//     Term 9 (APS4322-7000)/APS Outputs/Current Q 1X0 <-> Data Pointer/QCurrentSetPoints[6]
//     Term 9 (APS4322-7000)/APS Outputs/Current Q 1X1 <-> Data Pointer/QCurrentSetPoints[7]
//     Term 9 (APS4322-7000)/APS Outputs/Current Q 1X2 <-> Data Pointer/QCurrentSetPoints[8]
//     Term 9 (APS4322-7000)/APS Outputs/Current Q 2X0 <-> Data Pointer/QCurrentSetPoints[12]
//     Term 9 (APS4322-7000)/APS Outputs/Current Q 2X1 <-> Data Pointer/QCurrentSetPoints[13]
//     Term 9 (APS4322-7000)/APS Outputs/Current Q 2X2 <-> Data Pointer/QCurrentSetPoints[14]
//     Term 9 (APS4322-7000)/APS Outputs/Current Q 3X0 <-> Data Pointer/QCurrentSetPoints[18]
//     Term 9 (APS4322-7000)/APS Outputs/Current Q 3X1 <-> Data Pointer/QCurrentSetPoints[19]
//     Term 9 (APS4322-7000)/APS Outputs/Current Q 3X2 <-> Data Pointer/QCurrentSetPoints[20]
//     Term 9 (APS4322-7000)/APS Outputs/Current Q 0Y0 <-> Data Pointer/QCurrentSetPoints[3]
//     Term 9 (APS4322-7000)/APS Outputs/Current Q 0Y1 <-> Data Pointer/QCurrentSetPoints[4]
//     Term 9 (APS4322-7000)/APS Outputs/Current Q 0Y2 <-> Data Pointer/QCurrentSetPoints[5]
//     Term 9 (APS4322-7000)/APS Outputs/Current Q 1Y0 <-> Data Pointer/QCurrentSetPoints[9]
//     Term 9 (APS4322-7000)/APS Outputs/Current Q 1Y1 <-> Data Pointer/QCurrentSetPoints[10]
//     Term 9 (APS4322-7000)/APS Outputs/Current Q 1Y2 <-> Data Pointer/QCurrentSetPoints[11]
//     Term 9 (APS4322-7000)/APS Outputs/Current Q 2Y0 <-> Data Pointer/QCurrentSetPoints[15]
//     Term 9 (APS4322-7000)/APS Outputs/Current Q 2Y1 <-> Data Pointer/QCurrentSetPoints[16]
//     Term 9 (APS4322-7000)/APS Outputs/Current Q 2Y2 <-> Data Pointer/QCurrentSetPoints[17]
//     Term 9 (APS4322-7000)/APS Outputs/Current Q 3Y0 <-> Data Pointer/QCurrentSetPoints[21]
//     Term 9 (APS4322-7000)/APS Outputs/Current Q 3Y1 <-> Data Pointer/QCurrentSetPoints[22]
//     Term 9 (APS4322-7000)/APS Outputs/Current Q 3Y2 <-> Data Pointer/QCurrentSetPoints[23]
//     Term 9 (APS4322-7000)/APS Outputs/PhiE 0X0 <-> Data Pointer/PhiSetPoints[0]
//     Term 9 (APS4322-7000)/APS Outputs/PhiE 0X1 <-> Data Pointer/PhiSetPoints[1]
//     Term 9 (APS4322-7000)/APS Outputs/PhiE 0X2 <-> Data Pointer/PhiSetPoints[2]
//     Term 9 (APS4322-7000)/APS Outputs/PhiE 1X0 <-> Data Pointer/PhiSetPoints[6]
//     Term 9 (APS4322-7000)/APS Outputs/PhiE 1X1 <-> Data Pointer/PhiSetPoints[7]
//     Term 9 (APS4322-7000)/APS Outputs/PhiE 1X2 <-> Data Pointer/PhiSetPoints[8]
//     Term 9 (APS4322-7000)/APS Outputs/PhiE 2X0 <-> Data Pointer/PhiSetPoints[12]
//     Term 9 (APS4322-7000)/APS Outputs/PhiE 2X1 <-> Data Pointer/PhiSetPoints[13]
//     Term 9 (APS4322-7000)/APS Outputs/PhiE 2X2 <-> Data Pointer/PhiSetPoints[14]
//     Term 9 (APS4322-7000)/APS Outputs/PhiE 3X0 <-> Data Pointer/PhiSetPoints[18]
//     Term 9 (APS4322-7000)/APS Outputs/PhiE 3X1 <-> Data Pointer/PhiSetPoints[19]
//     Term 9 (APS4322-7000)/APS Outputs/PhiE 3X2 <-> Data Pointer/PhiSetPoints[20]
//     Term 9 (APS4322-7000)/APS Outputs/PhiE 0Y0 <-> Data Pointer/PhiSetPoints[3]
//     Term 9 (APS4322-7000)/APS Outputs/PhiE 0Y1 <-> Data Pointer/PhiSetPoints[4]
//     Term 9 (APS4322-7000)/APS Outputs/PhiE 0Y2 <-> Data Pointer/PhiSetPoints[5]
//     Term 9 (APS4322-7000)/APS Outputs/PhiE 1Y0 <-> Data Pointer/PhiSetPoints[9]
//     Term 9 (APS4322-7000)/APS Outputs/PhiE 1Y1 <-> Data Pointer/PhiSetPoints[10]
//     Term 9 (APS4322-7000)/APS Outputs/PhiE 1Y2 <-> Data Pointer/PhiSetPoints[11]
//     Term 9 (APS4322-7000)/APS Outputs/PhiE 2Y0 <-> Data Pointer/PhiSetPoints[15]
//     Term 9 (APS4322-7000)/APS Outputs/PhiE 2Y1 <-> Data Pointer/PhiSetPoints[16]
//     Term 9 (APS4322-7000)/APS Outputs/PhiE 2Y2 <-> Data Pointer/PhiSetPoints[17]
//     Term 9 (APS4322-7000)/APS Outputs/PhiE 3Y0 <-> Data Pointer/PhiSetPoints[21]
//     Term 9 (APS4322-7000)/APS Outputs/PhiE 3Y1 <-> Data Pointer/PhiSetPoints[22]
//     Term 9 (APS4322-7000)/APS Outputs/PhiE 3Y2 <-> Data Pointer/PhiSetPoints[23]
//     Term 9 (APS4322-7000)/Term 10 (APS4322-5000)/FB Inputs/A{0..8 step 2} X-Field <-> Data Pointer/HallSensorFieldsXYZ[{0..12 step 3}]  (5 links)
//     Term 9 (APS4322-7000)/Term 10 (APS4322-5000)/FB Inputs/A{0..8 step 2} Y-Field <-> Data Pointer/HallSensorFieldsXYZ[{1..13 step 3}]  (5 links)
//     Term 9 (APS4322-7000)/Term 10 (APS4322-5000)/FB Inputs/A{0..8 step 2} Z-Field <-> Data Pointer/HallSensorFieldsXYZ[{2..14 step 3}]  (5 links)
//     Term 9 (APS4322-7000)/Term 10 (APS4322-5000)/FB Inputs/B{1..9 step 2} X-Field <-> Data Pointer/HallSensorFieldsXYZ[{15..27 step 3}]  (5 links)
//     Term 9 (APS4322-7000)/Term 10 (APS4322-5000)/FB Inputs/B{1..9 step 2} Y-Field <-> Data Pointer/HallSensorFieldsXYZ[{16..28 step 3}]  (5 links)
//     Term 9 (APS4322-7000)/Term 10 (APS4322-5000)/FB Inputs/B{1..9 step 2} Z-Field <-> Data Pointer/HallSensorFieldsXYZ[{17..29 step 3}]  (5 links)
//     Term 9 (APS4322-7000)/Term 10 (APS4322-5000)/FB Inputs/C{0..8 step 2} X-Field <-> Data Pointer/HallSensorFieldsXYZ[{30..42 step 3}]  (5 links)
//     Term 9 (APS4322-7000)/Term 10 (APS4322-5000)/FB Inputs/C{0..8 step 2} Y-Field <-> Data Pointer/HallSensorFieldsXYZ[{31..43 step 3}]  (5 links)
//     Term 9 (APS4322-7000)/Term 10 (APS4322-5000)/FB Inputs/C{0..8 step 2} Z-Field <-> Data Pointer/HallSensorFieldsXYZ[{32..44 step 3}]  (5 links)
//     Term 9 (APS4322-7000)/Term 10 (APS4322-5000)/FB Inputs/D{1..9 step 2} X-Field <-> Data Pointer/HallSensorFieldsXYZ[{45..57 step 3}]  (5 links)
//     Term 9 (APS4322-7000)/Term 10 (APS4322-5000)/FB Inputs/D{1..9 step 2} Y-Field <-> Data Pointer/HallSensorFieldsXYZ[{46..58 step 3}]  (5 links)
//     Term 9 (APS4322-7000)/Term 10 (APS4322-5000)/FB Inputs/D{1..9 step 2} Z-Field <-> Data Pointer/HallSensorFieldsXYZ[{47..59 step 3}]  (5 links)
//     Term 9 (APS4322-7000)/Term 10 (APS4322-5000)/FB Inputs/E{0..8 step 2} X-Field <-> Data Pointer/HallSensorFieldsXYZ[{60..72 step 3}]  (5 links)
//     Term 9 (APS4322-7000)/Term 10 (APS4322-5000)/FB Inputs/E{0..8 step 2} Y-Field <-> Data Pointer/HallSensorFieldsXYZ[{61..73 step 3}]  (5 links)
//     Term 9 (APS4322-7000)/Term 10 (APS4322-5000)/FB Inputs/E{0..8 step 2} Z-Field <-> Data Pointer/HallSensorFieldsXYZ[{62..74 step 3}]  (5 links)
//     Term 9 (APS4322-7000)/Term 10 (APS4322-5000)/FB Inputs/F{1..9 step 2} X-Field <-> Data Pointer/HallSensorFieldsXYZ[{75..87 step 3}]  (5 links)
//     Term 9 (APS4322-7000)/Term 10 (APS4322-5000)/FB Inputs/F{1..9 step 2} Y-Field <-> Data Pointer/HallSensorFieldsXYZ[{76..88 step 3}]  (5 links)
//     Term 9 (APS4322-7000)/Term 10 (APS4322-5000)/FB Inputs/F{1..9 step 2} Z-Field <-> Data Pointer/HallSensorFieldsXYZ[{77..89 step 3}]  (5 links)
//     Term 9 (APS4322-7000)/Term 10 (APS4322-5000)/FB Inputs/G{0..8 step 2} X-Field <-> Data Pointer/HallSensorFieldsXYZ[{90..102 step 3}]  (5 links)
//     Term 9 (APS4322-7000)/Term 10 (APS4322-5000)/FB Inputs/G{0..8 step 2} Y-Field <-> Data Pointer/HallSensorFieldsXYZ[{91..103 step 3}]  (5 links)
//     Term 9 (APS4322-7000)/Term 10 (APS4322-5000)/FB Inputs/G{0..8 step 2} Z-Field <-> Data Pointer/HallSensorFieldsXYZ[{92..104 step 3}]  (5 links)
//     Term 9 (APS4322-7000)/Term 10 (APS4322-5000)/FB Inputs/H{1..9 step 2} X-Field <-> Data Pointer/HallSensorFieldsXYZ[{105..117 step 3}]  (5 links)
//     Term 9 (APS4322-7000)/Term 10 (APS4322-5000)/FB Inputs/H{1..9 step 2} Y-Field <-> Data Pointer/HallSensorFieldsXYZ[{106..118 step 3}]  (5 links)
//     Term 9 (APS4322-7000)/Term 10 (APS4322-5000)/FB Inputs/H{1..9 step 2} Z-Field <-> Data Pointer/HallSensorFieldsXYZ[{107..119 step 3}]  (5 links)
//     Term 9 (APS4322-7000)/Term 10 (APS4322-5000)/FB Inputs/I{0..8 step 2} X-Field <-> Data Pointer/HallSensorFieldsXYZ[{120..132 step 3}]  (5 links)
//     Term 9 (APS4322-7000)/Term 10 (APS4322-5000)/FB Inputs/I{0..8 step 2} Y-Field <-> Data Pointer/HallSensorFieldsXYZ[{121..133 step 3}]  (5 links)
//     Term 9 (APS4322-7000)/Term 10 (APS4322-5000)/FB Inputs/I{0..8 step 2} Z-Field <-> Data Pointer/HallSensorFieldsXYZ[{122..134 step 3}]  (5 links)
//     Term 9 (APS4322-7000)/Term 10 (APS4322-5000)/FB Inputs/J{1..9 step 2} X-Field <-> Data Pointer/HallSensorFieldsXYZ[{135..147 step 3}]  (5 links)
//     Term 9 (APS4322-7000)/Term 10 (APS4322-5000)/FB Inputs/J{1..9 step 2} Y-Field <-> Data Pointer/HallSensorFieldsXYZ[{136..148 step 3}]  (5 links)
//     Term 9 (APS4322-7000)/Term 10 (APS4322-5000)/FB Inputs/J{1..9 step 2} Z-Field <-> Data Pointer/HallSensorFieldsXYZ[{137..149 step 3}]  (5 links)
//     Term 9 (APS4322-7000)/Term 10 (APS4322-5000)/FB Inputs/Status <-> Data Pointer/FeedbackStatus

CONFIGURATION Plc
    RESOURCE PLC ON TwinCAT3
        TASK PlcTask(INTERVAL := T#10ms, PRIORITY := 6);
        PROGRAM MAIN WITH PlcTask : MAIN;
    END_RESOURCE
END_CONFIGURATION

// ---- THREADs/Example Product Data/ST_ProductDataA.TcDUT
TYPE ST_ProductDataA :
STRUCT
	nQuality : UINT;
	bGoodProduct : BOOL;
END_STRUCT
END_TYPE

// ---- THREADs/Example Product Data/I_ProductDataA.TcIO
INTERFACE I_ProductDataA EXTENDS I_XP_ProductData

{attribute 'monitoring':='call'}
PROPERTY Data : REFERENCE TO ST_ProductDataA
GET
END_GET
END_PROPERTY

END_INTERFACE

// ---- THREADs/MAIN.TcPOU
PROGRAM MAIN
VAR CONSTANT
	cCtsXpMovers : UINT := 3;	
	cCtsXpTracks : UINT := 6;	
	//Unique station identification 
	S_INFEED1 	: STRING := 'Station A';
	S_OUTFEED1 	: STRING := 'Station D';
	//Groupe station identification 
	G_PROCESS	: STRING := 'Groupe Process';
END_VAR
VAR
	bInitDone 			: BOOL;
	bEnable				: BOOL;
	bDisable, bReset	: BOOL;
	bSetSettings 		: BOOL := TRUE;
	
	(* XPlanar System - 1 per associated XPlanar 
		The system is the container and organizer for all subsequent XPlanar objects. All objects are registered with this system*)
	fbXpSystem : FB_XP_System;
	ipXPlanarPLC : I_XP_System_PLC := fbXpSystem; 
	
	(* XPlanar Collision Avoidance Groupe - 1 per associated XPlanar 
		The Planar group is a software object that prevents collisions between Planar movers as well as collisions of Planar movers with the boundary of 
		the stator area on the two-dimensional XPlanar stator area. To do this, the 2D areas of all objects in the group are blocked. When a motion command 
		is transferred to a mover, the required area is requested from the Planar group and the motion command is rejected if this area would collide 
		with already reserved areas. If the motion command can be executed, the area is added to the set of reserved area and blocked accordingly. *)
	fbXpGroup : FB_XP_Group
									(ipSystem			:= fbXpSystem);
	(* XPlanar Environment - 1 per associated XPlanar 
		The Planar environment is a software object that represents the two-dimensional XPlanar stator surface. Together with Planar movers in a group, 
		it prevents collisions of the movers with the edge of the surface. *)
	fbXpEnvironment : FB_XP_Environment
									(ipSystem			:= fbXpSystem);	
	
	(* XPlanar mover - n per associated XPlanar. Can be instantiated as an array and/or individually
		The Planar mover is a software object that represents an XPlanar mover. It summarizes the state of the real mover (position, velocity, etc.) 
		for the user. In addition, the user has the possibility to influence or control the state of the real mover via the Planar mover. *)								
	aMovers : ARRAY[1..cCtsXpMovers] OF FB_XP_Mover[
								 	(ipSystem			:= fbXpSystem),
								 	(ipSystem			:= fbXpSystem),
								 	(ipSystem			:= fbXpSystem)];

	(* XPlanar track - n per associated XPlanar. Can be instantiated as an array and/or individually
		The Planar track is a software object that represents a (virtual) one-dimensional path on the two-dimensional XPlanar stator surface. 
		Several Planar movers can be lined up and moved on this path. Collisions are prevented by keeping a preset distance between the movers. *)		
	aTracks : ARRAY[1..cCtsXpTracks] OF FB_XP_Track[
								 	(ipSystem			:= fbXpSystem),
								 	(ipSystem			:= fbXpSystem),
								 	(ipSystem			:= fbXpSystem),
								 	(ipSystem			:= fbXpSystem),
								 	(ipSystem			:= fbXpSystem),
								 	(ipSystem			:= fbXpSystem)];

	(* XPlanar station - n per associated XPlanar. Can be instantiated as an array and/or individually
		The stations are the main component of the application. As soon as the system has been started up and all movers are on the track, the movers are only sent from one station to the next.
		Parameters:
			xPos, yPos 			= Absolute position of the station on the xPlanar.
			ipAccocietedTrack 	= The track on which the station is located. If the XY position is not on this track, the next possible track position is assumed on this track.
								  Can be set to 0. In this case, the closest track to the coordinates is automatically used. 
								  If the station is very close to a transition, it may still be interesting to enter the exact track here.		
			sUniqueName 		= Unique name that may only exist once.
			sTargetGroup 		= A name for a group to which this station belongs. Important for redundant stations	*)	
	fbStationA : FB_XP_Station(ipSystem 			:= fbXpSystem,
									ipAccocietedTrack 	:= 0,// =closest track
									sUniqueName			:= S_INFEED1,
									sTargetGroup		:= '',
									nMoverQueueSize		:= 1,
									xPos				:= 100,
									yPos				:= 540);
									
	fbStationB 		: FB_XP_Station(ipSystem 			:= fbXpSystem,
									ipAccocietedTrack 	:= 0, // =closest track
									sUniqueName 		:= '',
									sTargetGroup		:= G_PROCESS,
									nMoverQueueSize		:= 1,
									xPos				:= 600,
									yPos				:= 600);	
		
	fbStationC 		: FB_XP_Station(ipSystem 			:= fbXpSystem,
									ipAccocietedTrack 	:= 0, // =closest track
									sUniqueName 		:= '',
									sTargetGroup		:= G_PROCESS,
									nMoverQueueSize		:= 1,
									xPos				:= 600,
									yPos				:= 120);						
										
	fbStationD 		: FB_XP_Station(ipSystem 			:= fbXpSystem,
									ipAccocietedTrack 	:= 0, // =closest track
									sUniqueName 		:= S_OUTFEED1,
									sTargetGroup		:= '',
									nMoverQueueSize		:= 2,
									xPos				:= 120,
									yPos				:= 400);	
											
	fbStationD_ChangeGap 		: FB_XP_Station(ipSystem := fbXpSystem,
									ipAccocietedTrack 	:= 0, // =closest track
									sUniqueName 		:= '',
									sTargetGroup		:= '',
									nMoverQueueSize		:= 1,
									xPos				:= 188,//120,125
									yPos				:= 90);						
													
	(*Processing station*)								
	fbStationCLowerZ : FB_Station_LowerZForce(ipStation := fbStationC);	
	fbStationBExternalSetpoint : FB_Station_ExternalSetpoint(ipStation := fbStationB);							
									
	(* EtherCAt diagnostics - TC3_Eventlogger
	This function block instance scans the entire EtherCat master. 
	Each EtherCat slave device is recognized and a message is written to the TC3_Eventlogger as soon as an unwanted state occurs.*)
	//	fbEtherCatDiagLAN3 : FB_EtherCatMasterDiag;
	//	fbEtherCatDiagLAN4 : FB_EtherCatMasterDiag;
END_VAR

//Example ConfigTrack
VAR
	bDoConfigTrackC 		: BOOL := TRUE;
	nSeqConfigTrack 		: UINT;
	fbTrackFeedback 		: MC_PlanarFeedback;	
	posStart, posEnd 		: PositionXYC; 
END_VAR

//Example SimulationMode
VAR
	bStartSimulation,bStopSimulation : BOOL;
END_VAR

//Example Manual Interaction with process outside XPlanar
VAR
	bToUpstreamProcessCanStart 		: BOOL; //Requestet cts of mover are in station. Example: rototer can start to place prodcts
	bFromUpsreamProcessIsFinish 	: BOOL; //The upstream process can set this bool if the process is finish and the mover can leave the station
	sFromUpstreamTagedStation		: STRING; //The Upstream can chose where the movers should go next
END_VAR

IF NOT bInitDone THEN
 	ipXPlanarPLC.Initialize();
	bInitDone := ipXPlanarPLC.Initialized;
	RETURN;
END_IF

IF bEnable AND ipXPlanarPLC.Disabled THEN
	bEnable := FALSE;
	ipXPlanarPLC.Enable();
	bSetSettings := TRUE; // Write Settings once
END_IF

IF bDisable OR bReset THEN
	bDisable := FALSE; bReset := FALSE;
	ipXPlanarPLC.Disable();
END_IF

IF bStartSimulation AND ipXPlanarPLC.Enabled THEN
	bStartSimulation := FALSE;
	fbStationA.SimulationStart(fProcessDuration := 0.1, sTargetStation := G_PROCESS); //Groupe
	fbStationD.SimulationStart(fProcessDuration := 0.5, sTargetStation := S_INFEED1); //Exact Station
	
	//fbStationB.SimulationStart(fProcessDuration := 1.0, sTargetStation := S_OUTFEED1); 
	fbStationBExternalSetpoint.TargetStation := S_OUTFEED1;	
	
	//fbStationC.SimulationStart(fProcessDuration := 1.0, sTargetStation := S_OUTFEED1);
	fbStationCLowerZ.TargetStation := S_OUTFEED1;
END_IF

IF bStopSimulation THEN
	bStopSimulation := FALSE;
	fbStationA.SimulationStop();
	fbStationB.SimulationStop();
	fbStationC.SimulationStop();
	fbStationD.SimulationStop();
END_IF


//Calculate setting each cycle
IF ipXPlanarPLC.Enabled THEN
	//Movement to the station is only permitted if the track is free. 
	//This serves to prevent collisions as only the gap is not sufficient here
	fbStationB.ReadyToRecvMovers := fbStationB.AccocietedTrack.CtsMoversOnTrack = 0;
	fbStationC.ReadyToRecvMovers := fbStationC.AccocietedTrack.CtsMoversOnTrack = 0;
ELSE
	fbStationB.ReadyToRecvMovers := FALSE;
	fbStationC.ReadyToRecvMovers := FALSE;
END_IF


//Do settings once at eanbling
IF bSetSettings THEN
	bSetSettings := FALSE;
	
	//TODO: The very first time the system is started up, the mover does not yet have a target. 
	//The default target defined in the CHALET_Xplanar/parameter list is entered. You should adjust the defaulttrged 

	//Set Mover Velocity, Acc, Dec, Jerk once. The station will override this settings
	aMovers[1].SetDynConstraint_Path(200,1900,1900,20000);
	aMovers[2].SetDynConstraint_Path(200,1900,1900,20000);
	aMovers[3].SetDynConstraint_Path(200,1900,1900,20000);
	
	//"In Position" is set 5mm earlier
	fbStationA.TargetPosWindow := 5.0;
	
	//The mover gets this targed gap asson he leves the station
	fbStationA.MoverGapAtExit := 300.0;
	fbStationD_ChangeGap.MoverGapAtExit := 190.0;
	
	fbStationB.MoverVelocityAtExit := 2000;	
	fbStationB.MoverAccAtExit := MC_MAXIMUM;
	fbStationB.MoverDecAtExit := MC_MAXIMUM;
	
	fbStationC.MoverVelocityAtExit := 2000;	
	fbStationC.MoverAccAtExit := MC_DEFAULT;
END_IF


PRG_Example_ProductData_Simple();


(* Update is called at the end of the program *)
ipXPlanarPLC.Update();
fbStationCLowerZ.Update();
fbStationBExternalSetpoint.Update();
//fbEtherCatDiagLAN3.Update();
//fbEtherCatDiagLAN4.Update();

METHOD Example_ManualConfigTrack : BOOL
(* Instead of the track being initialized in the track object, 
   the track progression can also be set here in the PLC. 
   To change values in the PLC, the track must be disabled (system is disabled) and the value to be changed must not be described in the object. 
*)
IF bDoConfigTrackC AND xPlanarPLC.Disabled THEN
	CASE nSeqConfigTrack OF
		0: //Clears the geometric information of the Planar Track.
			fbTrackC.PlanarTrack.Clear(fbTrackFeedback);
			nSeqConfigTrack := nSeqConfigTrack + 1;
		
		1: //Wait for command finished successfully
			IF fbTrackFeedback.Done THEN
				nSeqConfigTrack := nSeqConfigTrack + 1;
			END_IF
			
		2: //Sets the other Planar Tracks endpoint as start point of this Planar Track, transition is smooth. The other Planar Track is blocked for further changes (until it is cleared).
			fbTrackC.PlanarTrack.StartFromTrack(track := fbTrackA.PlanarTrack, commandFeedback := fbTrackFeedback);
			nSeqConfigTrack := nSeqConfigTrack + 1;
		
		3: //Wait for command finished successfully
			IF fbTrackFeedback.Done THEN
				nSeqConfigTrack := nSeqConfigTrack + 1;
			END_IF
			
		4: //Appends a line to the Planar Track.
			posStart.SetValuesXYC(840,480,0);
			posEnd.SetValuesXYC(840,240,0);
			fbTrackC.PlanarTrack.AppendLine(start := posStart, end := posEnd, commandFeedback := fbTrackFeedback);
			nSeqConfigTrack := nSeqConfigTrack + 1;					

		5: //Wait for command finished successfully
			IF fbTrackFeedback.Done THEN
				nSeqConfigTrack := nSeqConfigTrack + 1;
			END_IF
			
		6: //Appends a smooth transition from the end of this Planar Track to the other Planar Tracks start point. The Planar Track is blocked for further changes (until it is cleared).
			fbTrackC.PlanarTrack.EndAtTrack(track := fbTrackA.PlanarTrack, commandFeedback := fbTrackFeedback);
			nSeqConfigTrack := nSeqConfigTrack + 1;
		
		7: //Wait for command finished successfully
			IF fbTrackFeedback.Done THEN
				nSeqConfigTrack := nSeqConfigTrack + 1;
			END_IF		
		
		8: //Done
			bDoConfigTrackC := FALSE;
			nSeqConfigTrack := 0;
	END_CASE
	fbTrackFeedback.Update(); 
END_IF
END_METHOD

METHOD Example_ManualInteractionWithProcess : BOOL
(* Example: Interaction with process outside XPlanar 
   only works when the simulation is switched off
*)

//Requestet cts of mover are in station. Example: rototer can start to place prodcts
bToUpstreamProcessCanStart := xPlanarPLC.Station(S_INFEED1).MoversInPlace;

//The upstream process can set this bool if the process is finish and the mover can leave the station
bFromUpsreamProcessIsFinish := bFromUpsreamProcessIsFinish;

//The Upstream can chose where the movers should go next
//A group is specified here that contains several different. equivalent stations
sFromUpstreamTagedStation := G_OUTFEED;

IF bFromUpsreamProcessIsFinish AND bToUpstreamProcessCanStart AND xPlanarPLC.Enabled THEN
	bFromUpsreamProcessIsFinish := FALSE;
	xPlanarPLC.Station(S_INFEED1).SendMoversToStation(sFromUpstreamTagedStation);
END_IF
END_METHOD

END_PROGRAM

// ---- THREADs/FB_Station_LowerZForce.TcPOU
FUNCTION_BLOCK FB_Station_LowerZForce EXTENDS FB_CH_Object
VAR
	ipStation : I_XP_Station_PLC;
	nSeq : UINT;
	fbTon : TON;
	ipMoverInStation : I_XP_Mover_PLC;
	bFromUpstreamProcessIsFinish: BOOL := TRUE;
	sTargetStation : STRING; //the mover gets this as next target
END_VAR

METHOD FB_init : BOOL
VAR_INPUT
	bInitRetains : BOOL; // if TRUE, the retain variables are initialized (warm start / cold start)
	bInCopyCode : BOOL;  // if TRUE, the instance afterwards gets moved into the copy code (online change)
	
	ipStation : I_XP_Station_PLC;
	
END_VAR
VAR
	fbGetCurTaskIdx  : GETCURTASKINDEX;
END_VAR
THIS^.ipStation := ipStation;
END_METHOD

{attribute 'monitoring':='call'}
 //the mover gets this as next target
PROPERTY TargetStation : STRING
GET
TargetStation := sTargetStation;
END_GET
SET
sTargetStation := TargetStation;
END_SET
END_PROPERTY

METHOD Update : HRESULT
VAR
	refPlanarTrack : REFERENCE TO MC_PlanarTrack;
END_VAR
IF ipStation = 0 THEN
	RETURN; // ERROR
END_IF

IF ipStation.System.Disabled THEN
	nSeq := 0;
END_IF

//The simulation (automatic retransmission of a mover after a fixed time) is stopped for this station
ipStation.SimulationStop();

CASE nSeq OF 

	0: //wait for mover
		IF ipStation.MoversInPlace THEN
			//receive the foremost mover in the station (if there is more than one mover in the station)
			ipMoverInStation := ipStation.MoversInQueue[0];
			nSeq := 1;
		END_IF
		
	1: //Z = 0
		ipMoverInStation.LowerToUnknownLevel();
		nSeq := 2;				

	2: // wait until lowering is finish
		IF ipMoverInStation.Feedback.Done THEN
			fbTon.IN := FALSE;
			nSeq := 3;	
		END_IF
		
	3: //Delay 5s
		fbTon.IN := TRUE;
		IF fbTon.q THEN
			nSeq := 4;	
		END_IF			

	4: //Lift
		ipMoverInStation.LiftFromUnknownLevel();
		nSeq := 5;				

	5: // wait until lifting is finish
		//The upstream process can set this bool if the process is finish and the mover can leave the station
		bFromUpstreamProcessIsFinish := bFromUpstreamProcessIsFinish;

		fbTon.IN := TRUE;
		IF fbTon.q AND bFromUpstreamProcessIsFinish THEN
			nSeq := 100;	
		END_IF

		
	100: // send movers away to next target station or groupe. If no target exist, wait in this step
		IF sTargetStation <> '' THEN
			ipStation.SendMoversToStation(THIS^.sTargetStation);
			nSeq := 0;	
		END_IF

	
END_CASE
fbTon(PT:= T#5S);
END_METHOD

END_FUNCTION_BLOCK

// ---- THREADs/FB_Station_ExternalSetpoint.TcPOU
FUNCTION_BLOCK FB_Station_ExternalSetpoint EXTENDS FB_CH_Object
VAR
	ipStation : I_XP_Station_PLC;
	nSeq : UINT;
	fbTon : TON;
	ipMoverInStation : I_XP_Mover_PLC;
	bFromUpstreamProcessIsFinish: BOOL := TRUE;	
	sTargetStation : STRING; //the mover gets this as next target
END_VAR

METHOD FB_init : BOOL
VAR_INPUT
	bInitRetains : BOOL; // if TRUE, the retain variables are initialized (warm start / cold start)
	bInCopyCode : BOOL;  // if TRUE, the instance afterwards gets moved into the copy code (online change)
	
	ipStation : I_XP_Station_PLC;
	
END_VAR
THIS^.ipStation := ipStation;
END_METHOD

{attribute 'monitoring':='call'}
 //the mover gets this as next target
PROPERTY TargetStation : STRING
GET
TargetStation := sTargetStation;
END_GET
SET
sTargetStation := TargetStation;
END_SET
END_PROPERTY

METHOD Update : HRESULT
VAR
	fPositionOffsetX, fPositionOffsetY : LREAL;
END_VAR
IF ipStation = 0 THEN
	RETURN; // ERROR
END_IF

IF ipStation.System.Disabled THEN
	nSeq := 0;
END_IF

//The simulation (automatic retransmission of a mover after a fixed time) is stopped for this station
ipStation.SimulationStop();

CASE nSeq OF 
	0: //wait for mover
		IF ipStation.MoversInPlace THEN
			//receive the foremost mover in the station (if there is more than one mover in the station)
			ipMoverInStation := ipStation.MoversInQueue[0];
			IF ipMoverInStation <> 0 THEN
				nSeq := 1;
			END_IF
		END_IF
		
	1: //Switch on all external setpoint axes.
		ipMoverInStation.StartExternalSetpoint();
		nSeq := 2;				

	2: // wait until enabling is finish
		IF ipMoverInStation.Feedback.Done THEN
			fbTon.IN := FALSE;
			nSeq := 3;	
		END_IF
		
	3: //start Movement Example "scorrective movement" e.g.: a chamber has previously recognized the component and the tile must now align itself with this value
		ipMoverInStation.AxisExtSetpointX.MoveRelative(15,0,0,0,0,0);
		ipMoverInStation.AxisExtSetpointC.MoveRelative(-5,0,0,0,0,0);
		nSeq := 4;	
		
	4: 	//Wait for finish Movement
		//The upstream process can set this bool if the process is finish and the mover can leave the station
		bFromUpstreamProcessIsFinish := bFromUpstreamProcessIsFinish;
		IF ipMoverInStation.AxisExtSetpointX.Feedback.Done AND ipMoverInStation.AxisExtSetpointC.Feedback.Done AND bFromUpstreamProcessIsFinish THEN
			fbTon.IN := TRUE; //Start timer
			IF fbTon.Q THEN
				fbTon.IN := FALSE; //Reset timer
				nSeq := 5;					
			END_IF
		END_IF


	5: //Start Movement Example "exact station position" e.g.: The actual station is located slightly next to the track. It is particularly difficult to “hit” an exact position in the curve
		fPositionOffsetX := (ipStation.PositionXY.x - ipStation.PositionOnTrackXY.x);
		fPositionOffsetY := (ipStation.PositionXY.y - ipStation.PositionOnTrackXY.y);
		
		ipMoverInStation.AxisExtSetpointX.MoveAbsolute(fPosition := fPositionOffsetX,0,0,0,0,0);
		ipMoverInStation.AxisExtSetpointY.MoveAbsolute(fPosition := fPositionOffsetY,0,0,0,0,0);
		ipMoverInStation.AxisExtSetpointC.MoveAbsolute(fPosition := 0,0,0,0,0,0);
		nSeq := 6;	
		
	6: 	//Wait for finish Movement
		IF ipMoverInStation.AxisExtSetpointX.Feedback.Done AND ipMoverInStation.AxisExtSetpointY.Feedback.Done AND ipMoverInStation.AxisExtSetpointC.Feedback.Done THEN
			fbTon.IN := TRUE; //Start timer
			IF fbTon.Q THEN
				fbTon.IN := FALSE; //Reset timer
				nSeq := 7;					
			END_IF
		END_IF
	
	7: 	//Stop external Setpint
		ipMoverInStation.StopExternalSetpoint();
		nSeq := 8;	

	8: // wait until enable is finish
		IF ipMoverInStation.Feedback.Done THEN
			fbTon.IN := FALSE;
			nSeq := 100;	
		END_IF
		
	100: // send movers away to next target station or groupe. If no target exist, wait in this step
		IF sTargetStation <> '' THEN
			ipStation.SendMoversToStation(THIS^.sTargetStation);
			nSeq := 0;	
		END_IF	
	
END_CASE

fbTon(PT:= T#1S);
END_METHOD

END_FUNCTION_BLOCK

// ---- THREADs/Example Product Data/PRG_Example_ProductData_Simple.TcPOU
PROGRAM PRG_Example_ProductData_Simple
VAR
	bInitDone : BOOL;
		
	aProductsFormatA 		: ARRAY[1..MAIN.cCtsXpMovers] OF FB_ProductDataA;
	ipMover					: I_XP_Mover_PLC;
	ipProductDataOnMover 	: I_ProductDataA;
	ipStationModify 		: I_XP_Station_PLC;
	fbTriggerMoverInPlace 	: R_TRIG; 
	
	nIdx : DINT;
END_VAR

(* This example shows how easy it is to access the product data on the Mover. 
   The structure "ST_ProductDataA" can be edited to change the contained data.
*)

//Do this once during initialization
IF NOT bInitDone THEN
	bInitDone := TRUE;
	
	//A separate FB with product data is added to each mover
	FOR nIdx := 1 TO MAIN.cCtsXpMovers DO
		ipMover := MAIN.aMovers[nIdx]; 
		ipMover.ProductData := aProductsFormatA[nIdx];
	END_FOR
END_IF



//Get interface to StationB
ipStationModify := MAIN.ipXPlanarPLC.Station(MAIN.S_INFEED1);
IF ipStationModify = 0 THEN
	//Abort, Station is unknown
	RETURN;
END_IF

//This is executed once when the mover arrives at the station
fbTriggerMoverInPlace(CLK:= ipStationModify.MoversInPlace);
IF fbTriggerMoverInPlace.Q THEN
	
	//Do this for each mover inside the station
	FOR nIdx := 0 TO (ipStationModify.MoverQueueSize-1) DO
		
		//Query whether the FB behind this instance implements the following interface and get it.
		IF __QUERYINTERFACE(ipStationModify.MoversInQueue[nIdx].ProductData, ipProductDataOnMover) THEN 
			//Modify data. read and write
			ipProductDataOnMover.Data.nQuality 		:= ((ipProductDataOnMover.Data.nQuality + 42)MOD 100);	
			ipProductDataOnMover.Data.bGoodProduct 	:= ipProductDataOnMover.Data.nQuality >= 80;
			//ipProductDataOnMover. ...
		END_IF
	
	END_FOR
END_IF

END_PROGRAM

// ---- THREADs/FB_Station_Disable.TcPOU
FUNCTION_BLOCK FB_Station_Disable EXTENDS FB_CH_Object
VAR
	ipStation : I_XP_Station_PLC;
	sTargetStation : STRING; //the mover gets this as next target
END_VAR

METHOD FB_init : BOOL
VAR_INPUT
	bInitRetains : BOOL; // if TRUE, the retain variables are initialized (warm start / cold start)
	bInCopyCode : BOOL;  // if TRUE, the instance afterwards gets moved into the copy code (online change)
	
	ipStation : I_XP_Station_PLC;
	
END_VAR
VAR
	fbGetCurTaskIdx  : GETCURTASKINDEX;
END_VAR
THIS^.ipStation := ipStation;
END_METHOD

{attribute 'monitoring':='call'}
 //the mover gets this as next target
PROPERTY TargetStation : STRING
GET
TargetStation := sTargetStation;
END_GET
SET
sTargetStation := TargetStation;
END_SET
END_PROPERTY

METHOD Update : HRESULT
VAR
	refPlanarTrack : REFERENCE TO MC_PlanarTrack;
END_VAR

VAR_INST
	nSeq : UINT;
	fbFeedback : MC_PlanarFeedback;
	fbTon : TON;
	ipMoverInStation : I_XP_Mover_PLC;
END_VAR
IF ipStation = 0 THEN
	RETURN; // ERROR
END_IF

IF ipStation.System.Disabled THEN
	nSeq := 0;
END_IF

ipStation.SimulationStop();

CASE nSeq OF 

	0: //wait for mover
		IF ipStation.MoversInPlace THEN
			ipMoverInStation := ipStation.MoversInQueue[0];
			nSeq := 1;
		END_IF
		
	1: //disable
		ipMoverInStation.PlanarMover.Disable(fbFeedback);
		nSeq := 2;				

	2: // wait until disable is finish
		IF fbFeedback.Done THEN
			fbTon.IN := FALSE;
			nSeq := 3;	
		END_IF
		
	3: //Delay 5s
		fbTon.IN := TRUE;
		IF fbTon.q THEN
			nSeq := 4;	
		END_IF			

	4: //enable
		ipMoverInStation.PlanarMover.Enable(fbFeedback);
		nSeq := 5;				

	5: // wait until enable is finish
		IF fbFeedback.Done THEN
			fbTon.IN := FALSE;
			nSeq := 6;	
		END_IF
		
	6: //join Track
		refPlanarTrack REF= ipStation.AccocietedTrack.PlanarTrack;
		ipMoverInStation.PlanarMover.JoinTrack(	commandFeedback	:= fbFeedback, 
												targetTrack		:= refPlanarTrack, 
												constraint		:= ipMoverInStation.DynConstraint, 
												options			:= 0);
		nSeq := 7;				

	7: // wait until enable is finish
		IF fbFeedback.Done THEN
			fbTon.IN := FALSE;
			nSeq := 8;	
		END_IF
		
	8: // send movers away
		ipStation.SendMoversToStation(THIS^.sTargetStation);
		nSeq := 0;	
	
END_CASE
fbFeedback.Update();
fbTon(PT:= T#5S);
END_METHOD

END_FUNCTION_BLOCK
